FUNCTION_BLOCK FB_Tank
VAR_INPUT
END_VAR
VAR_OUTPUT
END_VAR
VAR
	_rCurrentLevel	: REAL;
	_rMaxCapacity	: REAL;	
	_bIsEmpty		: BOOL;

	bAlarmNextCycle	: BOOL;		//ADDITIONAL VARIABLE TO STOP PUMP BEFORE OVERFLOWING
END_VAR

PROPERTY bIsEmpty : BOOL
GET
//EMPTY WHEN CURRENT LEVEL IS 0
bIsEmpty	:= rCurrentLevel = 0.0;
END_GET
SET
END_SET
END_PROPERTY

PROPERTY bLevelHigh : BOOL
GET
//LEVEL IS HIGH IF CURRENT LEVEL IS EQUAL TO TANK MAX CAPACITY OR OVERFLOATING IN NEXT CYCLE
bLevelHigh	:= (rCurrentLevel = rMaxCapacity) OR bAlarmNextCycle;
END_GET
SET
END_SET
END_PROPERTY

PROPERTY bLevelLow : BOOL
GET
VAR
END_VAR
VAR CONSTANT
	LOW_LVL_TRESHOLD		: REAL := 1.0;		//LITER
END_VAR
bLevelLow	:= rCurrentLevel < LOW_LVL_TRESHOLD;
END_GET
SET
END_SET
END_PROPERTY

METHOD FB_init : BOOL
VAR_INPUT
	bInitRetains : BOOL; // if TRUE, the retain variables are initialized (warm start / cold start)
	bInCopyCode : BOOL;  // if TRUE, the instance afterwards gets moved into the copy code (online change)
END_VAR
//INITIALIZE TANK MAX CAPACITY
rMaxCapacity	:= 1000;
END_METHOD

PROPERTY rCurrentLevel : REAL
GET
rCurrentLevel	:= _rCurrentLevel;
END_GET
SET
_rCurrentLevel	:= rCurrentLevel;
END_SET
END_PROPERTY

METHOD Reset : BOOL
VAR_INPUT
END_VAR
//SET CURRENT TANK LEVEL TO 0
rCurrentLevel		:= 0.0;
END_METHOD

PROPERTY rMaxCapacity : REAL
GET
rMaxCapacity	:= _rMaxCapacity;
END_GET
SET
_rMaxCapacity	:= rMaxCapacity;
END_SET
END_PROPERTY

METHOD SetCapacity : BOOL
VAR_INPUT
	rCapacity		: REAL;
END_VAR
//SET CAPACITY
rMaxCapacity	:= rCapacity;
END_METHOD

METHOD UpdateLevel : BOOL
VAR_INPUT
	rFlowRate		: REAL;
	rTimeStepSec	: REAL;
END_VAR
VAR
	rCyclicLvlChange	: REAL;
END_VAR
(*1. CALCULATE NEW LEVEL*)
	rCyclicLvlChange	:= rFlowRate * rTimeStepSec;
	rCurrentLevel		:= rCurrentLevel + rCyclicLvlChange;

(*2. STOP IF OVERFLOWING IN NEXT CYCLE*)
	IF rCurrentLevel + rCyclicLvlChange > rMaxCapacity THEN
		bAlarmNextCycle		:= TRUE;
	ELSE
		bAlarmNextCycle		:= FALSE;
	END_IF
	
(*3. EMPTYING*)
	IF rCurrentLevel < 0 THEN
		Reset();
	END_IF
END_METHOD

END_FUNCTION_BLOCK

(* stored: Version 1.1.0.1, ProductVersion 3.1.4024.12
   POU FB_Tank: Id {bd8d5336-68c0-445e-a07c-065a6d58a3d0}, SpecialFunc None
   Property bIsEmpty: Id {a33a96fc-6dea-4582-858a-ae788a215348}
   Get Get: Id {17dbde76-0a2c-40f4-9295-e769ba6dd2f5}
   Set Set: Id {33671045-3fdc-4f96-9f86-c61d4b07067f}
   Property bLevelHigh: Id {88b91fe1-67e7-4349-b933-fd8b97a40b40}
   Get Get: Id {7e8217f0-9721-472b-89cc-03b5f2dea8fa}
   Set Set: Id {e5bfd86d-b43d-4a2a-82cd-4b0f2ad1891c}
   Property bLevelLow: Id {8e2ff05e-bebc-437f-890f-a483a51701c4}
   Get Get: Id {d379d92f-ee9f-4411-a72f-eb46c5bf4274}
   Set Set: Id {dca4beac-d453-4225-9d1e-d8caa9bd112f}
   Method FB_init: Id {b31aa727-c80d-4011-bcac-dcd4f8893590}
   Property rCurrentLevel: Id {4ded2a91-2be9-4894-abd6-2aa0b71038e1}
   Get Get: Id {a201ff39-d994-43d8-8d7b-e66f1691022e}
   Set Set: Id {b2586ac1-cbaa-4841-b880-7e084f102cf1}
   Method Reset: Id {e8edc8f3-e863-44e6-a1f9-389c830a11c2}
   Property rMaxCapacity: Id {5a210318-22fb-4956-a99b-2203242e72f9}
   Get Get: Id {467db33c-1768-42b0-9229-bcb9847f14db}
   Set Set: Id {b833c552-a9fc-4e86-bff6-6a18911e7707}
   Method SetCapacity: Id {bdd53ec9-e7e3-4b3e-ab54-efe4e67e1e89}
   Method UpdateLevel: Id {7e8cdd2d-27e8-480c-8d35-a624e933cd0d} *)
